{attribute 'qualified_only'}
VAR_GLOBAL RETAIN
	//Brauchwassermenge verbraucht in m3
    waterConsumption : WORD;
	waterConsumptionZisterne : WORD;
END_VAR

(* stored: Version 1.1.0.1, ProductVersion 3.1.4024.4
   GVL gvl_RETAIN: Id {81896dc9-140d-488f-8703-0c7f43325d42} *)
